Universal Robots PolyScope program: matlab_rsa_3.3.urp

Program matlab_rsa (createdIn=1.8.11657.0 lastSavedIn=3.3.4.310 directory=/programs/usbdisk installation=default robotSerialNumber=2017353993)
Calibrated DH parameters: a=[0.000164, -0.372614, -0.390071, 0.000067, 0.000035, 0]; d=[0.088949, -236.832261, 239.457522, -2.515251, 0.094878, 0.082509]; alpha=[1.570462, -0.000861, -0.0155, 1.570767, -1.57079, 0]; deltaTheta=[0.000015, 0.500831, -0.604847, 0.10386, 0.000033, 0.000067]
BeforeStart
  var_safety := 1
  var_safety_forc := 50
  var_moveType := [1,0]
  receive_data := [6,0,0,0,0,0,0]
  Move_To_Pos := p[0,0,0,0,0,0]
  var_moving := 0
  Call pgr_setupPose
  SuppressedNode
    receive_data := [5,110,0,40,0,40]
  ''
  SuppressedNode
    Call p08_setRG2
  var_velacc := [0.2,0.2]
  SuppressedNode
    Script: socket_open("192.168.10.2",30000)
  Script: socket_open("172.20.13.30",30000)
  task := [0,0]
  coop := 0
Robot Program (runOnlyOnce=false motionType=MoveJ speed=1.047198 acceleration=1.396263 recalculateMotions=false)
  SuppressedNode
    MoveJ speed 60 deg/s, acceleration 80 deg/s^2 (recalculateMotions=false)
      Waypoint Waypoint_1 (Relative): relativeFromPosition TCP in base x=416.871 y=-406.97 z=211.075 mm, rx=1.6627 ry=-1.7508 rz=0.7521 rad; joints [-27.823, -125.587, -73.499, -225.375, -46.749, 144.79] deg; TCP in base x=416.871 y=-406.97 z=211.075 mm, rx=1.6627 ry=-1.7508 rz=0.7521 rad; joints [-27.823, -125.587, -73.499, -225.375, -46.749, 144.79] deg; flange x=416.094 y=-405.791 z=208.632 mm, rx=1.6655 ry=-1.766 rz=0.7464 rad
  SuppressedNode
    coop := 1
  SuppressedNode
    Wait Sleep waitTime=2
  SuppressedNode
    coop := 0
  Script: task=socket_read_ascii_float(1)
  Wait Sleep waitTime=0.01
  If task[1]≟2
    Call p02_readPosC
    task := [0,0]
  ElseIf task[1]≟93
    coop := 1
    Script: socket_send_string("1")
    task := [0,0]
  ElseIf task[1]≟94
    coop := 0
    Script: socket_send_string("1")
    task := [0,0]
  ElseIf task[1]≟5
    Call p05_setIO
  ElseIf task[1]≟6
    Call p06_setMovement
  ElseIf task[1]≟7
    Call p07_SetVelAcc
  ElseIf task[1]≟8
    Call p08_setRG2
  ElseIf task[1]≟9
    Call p09_readDigital
  ElseIf task[1]≟10
    Call p10_readAnalog
  ElseIf task[1]≟1
    Call p01_move
SubProgram Safety_Program (keepSynchronizedWithDisk=false trackProgramExecution=false)
  var_safety := 0
  MoveJ speed 60 deg/s, acceleration 80 deg/s^2 (recalculateMotions=false)
    Waypoint safety_move_rel (Relative): motionParameters(jointSpeed=0.10472 jointAcceleration=1.396263 cartesianSpeed=0.25 cartesianAcceleration=1.2); relativeFromPosition TCP in base x=-200 y=-199.982 z=199.995 mm, rx=-3.1416 ry=0.0001 rz=0 rad; joints [-112.3, -58.235, -115.648, -96.117, 90, -202.3] deg; TCP in base x=-197.452 y=-201.523 z=235.542 mm, rx=3.1363 ry=0.0005 rz=0.0212 rad; joints [-112.312, -58.281, -115.231, -96.487, 90, -202.306] deg; flange x=-199.804 y=-200.621 z=410.561 mm, rx=3.1362 ry=0.0006 rz=0.0211 rad
    Wait Sleep waitTime=1
  Script: socket_send_string("2")
Thread Thread_1 (runOnlyOnce=false trackProgramExecution=false)
  If coop≟1
    Loop While (checkContinuously=false) expression=coop≟1
      Force Frame feature=Base; selection=[1, 1, 1, 1, 1, 1]; wrench=[0, 0, 0, 0, 0, 0]; limitsForce=[0.15, 0.15, 0.15, 1.047198, 1.047198, 1.047198]; limitsMotion=[0.1, 0.1, 0.1, 0.174533, 0.174533, 0.174533]
        Wait Sleep waitTime=0.01
    coop := 0
    Call pgr_setupPose
  Else 
    SuppressedNode
      Script: movel(Move_To_Pos,a=var_velacc[0],v=var_velacc[1],r=0)
    If force()<var_safety_forc (checkContinuously=true)
      If var_moving≟1
        If var_safety≟1
          If var_moveType[0]≟1
            Script: movel(Move_To_Pos,a=var_velacc[0],v=var_velacc[1],r=0)
            If pose_dist(get_forward_kin(),Move_To_Pos)<0.01
              Script: socket_send_string("1")
              var_moving := 0
          Else 
            Script: movej(Move_To_Pos,a=var_velacc[0],v=var_velacc[1],r=0)
            If pose_dist(Base,Move_To_Pos)<0.01
              Script: socket_send_string("1")
              var_moving := 0
    Else 
      Call Safety_Program
    cur_velvac := var_velacc
    Wait Sleep waitTime=0.01
SubProgram -> pgr_setupPose
SubProgram -> p01_move
SubProgram -> p02_readPosC
SubProgram p03_readPosJ (keepSynchronizedWithDisk=false trackProgramExecution=false)
  Script: pose_1=get_actual_joint_positions()
  Script: socket_send_string(pose_1)
SubProgram -> p05_setIO
SubProgram -> p06_setMovement
SubProgram -> p07_SetVelAcc
SubProgram -> p08_setRG2
SubProgram -> p09_readDigital
SubProgram -> p10_readAnalog
SubProgram pgr_setupPose (keepSynchronizedWithDisk=false trackProgramExecution=false)
  Script: pose_1=get_forward_kin()
  pointer := 0
  Loop While (checkContinuously=false) expression=pointer<receive_data[0]
    Script: Move_To_Pos[pointer]=pose_1[pointer]
    pointer := pointer+1
SubProgram p08_setRG2 (keepSynchronizedWithDisk=false trackProgramExecution=false)
  'Set parameters for OnRobot RG2 gripper'
  Script: receive_data=socket_read_ascii_float(6)
  If receive_data[0]≠6
    Script: socket_send_string("0")
  Else 
    Script: socket_send_string("1")
    DO8_Off_DO9_Off := receive_data[1]
    DO8_On_DO9_Off := receive_data[2]
    DO8_Off_DO9_On := receive_data[3]
    DO8_On_DO9_On := receive_data[4]
    Grip_Force := receive_data[5]
    Script file /home/ur/ursim-3.0/programs/R1 04-01-2015/Release1.00-04-01-2015/Technical scripts/wrap1G4P1F.txt
      | if Grip_Force > 40:
      | 	Grip_Force = 40
      | 	popup("'Grip_Force' is too high - the value have been limited to  40N", title="Warning",  warning = True, error=False)
      | 	pause
      | end
      | 
      | if Grip_Force < 3:
      | 	Grip_Force = 3
      | 	popup("'Grip_Force' is too low - the value have been limited to  3N", title="Warning",  warning = True, error=False)
      | 	pause
      | end
      | 
      | if DO8_Off_DO9_Off > 110:
      | 	DO8_Off_DO9_Off = 110
      | 	popup("'DO8_Off_DO9_Off ' is too high - the value have been limited to  110mm", title="Warning",  warning = True, error=False)
      | 	pause
      | end
      | 
      | if DO8_Off_DO9_Off < 0:
      | 	DO8_Off_DO9_Off = 0
      | 	popup("'DO8_Off_DO9_Off ' is too low - the value have been limited to  0mm", title="Warning",  warning = True, error=False)
      | 	pause
      | end
      | 
      | if DO8_Off_DO9_On > 110:
      | 	DO8_Off_DO9_On = 110
      | 	popup("'DO8_Off_DO9_On ' is too high - the value have been limited to  110mm", title="Warning",  warning = True, error=False)
      | 	pause
      | end
      | 
      | if DO8_Off_DO9_On < 0:
      | 	DO8_Off_DO9_On = 0
      | 	popup("'DO8_Off_DO9_On ' is too low - the value have been limited to  0mm", title="Warning",  warning = True, error=False)
      | 	pause
      | end
      | 
      | 
      | 
      | 
      | if DO8_On_DO9_Off > 110:
      | 	DO8_On_DO9_Off = 110
      | 	popup("'DO8_On_DO9_Off ' is too high - the value have been limited to  110mm", title="Warning",  warning = True, error=False)
      | 	pause
      | end
      | 
      | if DO8_On_DO9_Off < 0:
      | 	DO8_On_DO9_Off = 0
      | 	popup("'DO8_On_DO9_Off ' is too low - the value have been limited to  0mm", title="Warning",  warning = True, error=False)
      | 	pause
      | end
      | 
      | if DO8_On_DO9_On > 110:
      | 	DO8_On_DO9_On = 110
      | 	popup("'DO8_On_DO9_On ' is too high - the value have been limited to  110mm", title="Warning",  warning = True, error=False)
      | 	pause
      | end
      | 
      | if DO8_On_DO9_On < 0:
      | 	DO8_On_DO9_On = 0
      | 	popup("'DO8_On_DO9_On ' is too low - the value have been limited to  0mm", title="Warning",  warning = True, error=False)
      | 	pause
      | end
      | 
      | 
      | #simple mapping
      | force0 = floor(Grip_Force)
      | pos0 = floor(DO8_On_DO9_On*10)
      | force1 = floor(Grip_Force)
      | pos1 = floor(DO8_Off_DO9_On*10)
      | force2 = floor(Grip_Force)
      | pos2 = floor(DO8_On_DO9_Off*10)
      | force3 = floor(Grip_Force)
      | pos3 = floor(DO8_Off_DO9_Off*10)
    Script file /home/ur/ursim-3.0/programs/R1 04-01-2015/Script update 1.01/Technical scripts/program_gripper.txt
      | def bit_bang_spi_master_UR_script(input):
      | 	local i = 0
      | 	while i < 8:
      | 		set_digital_out(8, True)
      | 
      | 		if input >= 128:
      | 			set_digital_out(9, False)
      | 			input = input - 128
      | 		 else:
      | 		  	set_digital_out(9, True)
      | 		  end
      | 		  input = input * 2
      | 		  sleep(0.008)
      | 		  set_digital_out(8, False)
      | 		  sleep(0.008)
      | 		  i = i + 1
      |   	end
      | end
      | 
      | 
      | 
      | version_number = 0
      | length = 15
      | 
      | set_digital_out(9, False)
      | set_digital_out(8, False)
      | set_tool_voltage(0)
      | sleep(1.5)
      | set_tool_voltage(24)
      | sleep(0.032)
      | set_tool_voltage(0)
      | sleep(0.064)
      | 
      | set_tool_voltage(24)
      | sleep(0.032)
      | set_tool_voltage(0)
      | sleep(0.064)
      | 
      | set_tool_voltage(24)
      | sleep(0.032)
      | set_tool_voltage(0)
      | sleep(0.064)
      | 
      | set_tool_voltage(24)
      | sleep(0.032)
      | set_tool_voltage(0)
      | sleep(0.064)
      | 
      | set_tool_voltage(24)
      | 
      | 
      | timeout = 0
      | while get_digital_in(8) == False:
      | 	timeout = timeout+1
      | 	sleep(0.008)
      | 	if timeout > 250:
      | 		popup("Gripper is not responding", title="Error",  warning = False, error=True)
      | 		return 1
      | 	end
      | end
      | 
      | 
      | 
      | timeout = 0
      | while get_digital_in(9):
      | 	timeout = timeout+1
      | 	sleep(0.008)
      | 	if timeout > 250:
      | 		popup("Gripper is not responding", title="Error",  warning = False, error=True)
      | 		return 1
      | 	end
      | end
      | 
      | 
      | bit_bang_spi_master_UR_script(version_number)
      | bit_bang_spi_master_UR_script(length)
      | 
      | bit_bang_spi_master_UR_script(force0)
      | bit_bang_spi_master_UR_script(pos0 - (floor(pos0/256)*256))
      | bit_bang_spi_master_UR_script(floor(pos0/256))
      | 
      | bit_bang_spi_master_UR_script(force1)
      | bit_bang_spi_master_UR_script(pos1 - (floor(pos1/256)*256))
      | bit_bang_spi_master_UR_script(floor(pos1/256))
      | 
      | bit_bang_spi_master_UR_script(force2)
      | bit_bang_spi_master_UR_script(pos2 - (floor(pos2/256)*256))
      | bit_bang_spi_master_UR_script(floor(pos2/256))
      | 
      | bit_bang_spi_master_UR_script(force3)
      | bit_bang_spi_master_UR_script(pos3 - (floor(pos3/256)*256))
      | bit_bang_spi_master_UR_script(floor(pos3/256))
      | 
      | bit_bang_spi_master_UR_script(85)
      | 
      | 
      | 
      | set_digital_out(9, False)
      | set_digital_out(8, False)
      | 
      | timeout = 0
      | while get_digital_in(9) == True:
      | 	timeout = timeout+1
      | 	sleep(0.008)
      | 	if timeout > 250:
      | 		popup("Gripper is not responding", title="Error",  warning = False, error=True)
      | 		return 1
      | 	end
      | end
      | 
      | timeout = 0
      | while get_digital_in(9) == False:
      | 	timeout = timeout+1
      | 	sleep(0.008)
      | 	if timeout > 250:
      | 		popup("Gripper is not responding", title="Error",  warning = False, error=True)
      | 		return 1
      | 	end
      | end
      | 
      | return 0
    task := [0,0]
SubProgram p02_readPosC (keepSynchronizedWithDisk=false trackProgramExecution=false)
  'Read pose'
  Script: pose_1=get_forward_kin()
  Script: socket_send_string(pose_1)
SubProgram p05_setIO (keepSynchronizedWithDisk=false trackProgramExecution=false)
  'Set I/O params'
  Script: receive_data=socket_read_ascii_float(6)
  If receive_data[0]≠6
    Script: socket_send_string("0")
  Else 
    Script: socket_send_string("1")
    If receive_data[1]≟ True
      Script: digital_out[receive_data[2]]= True
    Else 
      Script: digital_out[receive_data[2]]= False
    task := [0,0]
SubProgram p06_setMovement (keepSynchronizedWithDisk=false trackProgramExecution=false)
  'Set movement type'
  Script: receive_data=socket_read_ascii_float(6)
  If receive_data[0]≠6
    Script: socket_send_string("0")
  Else 
    Script: socket_send_string("1")
    If receive_data[1]≟1
      var_moveType := [1,0]
    Else 
      var_moveType := [2,0]
SubProgram p07_SetVelAcc (keepSynchronizedWithDisk=false trackProgramExecution=false)
  'velocity and acceleration parameters'
  Script: receive_data=socket_read_ascii_float(6)
  If receive_data[0]≠6
    Script: socket_send_string("0")
  Else 
    Script: socket_send_string("1")
    pointer := 0
    Loop While (checkContinuously=false) expression=pointer<receive_data[0]
      Script: var_velacc[pointer]=receive_data[pointer+1]
      pointer := pointer+1
    task := [0,0]
SubProgram p09_readDigital (keepSynchronizedWithDisk=false trackProgramExecution=false)
  Script: receive_data=socket_read_ascii_float(2)
  If receive_data[0]≠2
    Script: socket_send_string("0")
  Else 
    Script: socket_send_string("1")
    Wait Sleep waitTime=0.01
    If digital_in[receive_data[1]] ≟ True
      Script: socket_send_string("1")
    Else 
      Script: socket_send_string("0")
    task := [0,0]
SubProgram p10_readAnalog (keepSynchronizedWithDisk=false trackProgramExecution=false)
  Script: receive_data=socket_read_ascii_float(2)
  If receive_data[0]≠2
    Script: socket_send_string("0")
  Else 
    Script: socket_send_string("1")
    Wait Sleep waitTime=0.01
    Script: socket_send_string( analog_in[receive_data[1]] )
    task := [0,0]
SubProgram p01_move (keepSynchronizedWithDisk=false trackProgramExecution=false)
  'robot position and orientation'
  Script: receive_data=socket_read_ascii_float(6)
  If receive_data[0]≠6
    Script: socket_send_string("0")
  Else 
    Script: socket_send_string("1")
    pointer := 0
    Loop While (checkContinuously=false) expression=pointer<receive_data[0]
      Script: Move_To_Pos[pointer]=receive_data[pointer+1]
      pointer := pointer+1
    var_moving := 1
    task := [0,0]
